// TIA Portal V19 export
FUNCTION_BLOCK "StatusSummary"   // FB63, F_FBD
TITLE = StatusSummary
AUTHOR : Siemens AG DI FA S SUP
// Summarize the Status Information from all Safety Zones and form general diagnostic bits.
// stored: Namespace Safety
   VAR_IN_OUT
      status : "Safety.typeDataFromSafety";
   END_VAR
BEGIN

REGION Network 1: Summarize Estop Functions
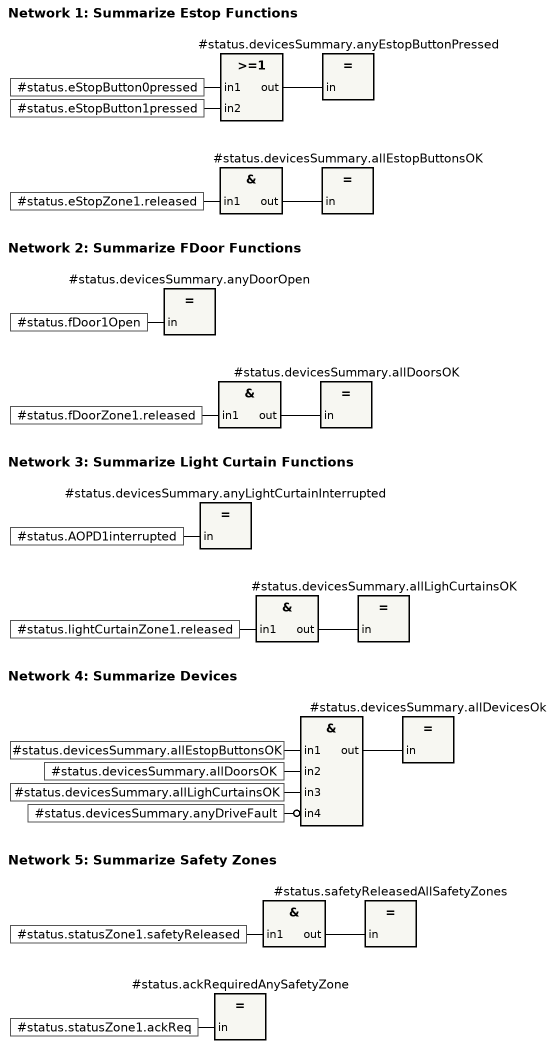
   #status.devicesSummary.anyEstopButtonPressed := #status.eStopButton0pressed OR #status.eStopButton1pressed;
   #status.devicesSummary.allEstopButtonsOK := #status.eStopZone1.released;
END_REGION

REGION Network 2: Summarize FDoor Functions
   #status.devicesSummary.anyDoorOpen := #status.fDoor1Open;
   #status.devicesSummary.allDoorsOK := #status.fDoorZone1.released;
END_REGION

REGION Network 3: Summarize Light Curtain Functions
   #status.devicesSummary.anyLightCurtainInterrupted := #status.AOPD1interrupted;
   #status.devicesSummary.allLighCurtainsOK := #status.lightCurtainZone1.released;
END_REGION

REGION Network 4: Summarize Devices
   #status.devicesSummary.allDevicesOk := #status.devicesSummary.allEstopButtonsOK AND #status.devicesSummary.allDoorsOK AND #status.devicesSummary.allLighCurtainsOK AND NOT #status.devicesSummary.anyDriveFault;
END_REGION

REGION Network 5: Summarize Safety Zones
   #status.safetyReleasedAllSafetyZones := #status.statusZone1.safetyReleased;
   #status.ackRequiredAnySafetyZone := #status.statusZone1.ackReq;
END_REGION
END_FUNCTION_BLOCK
